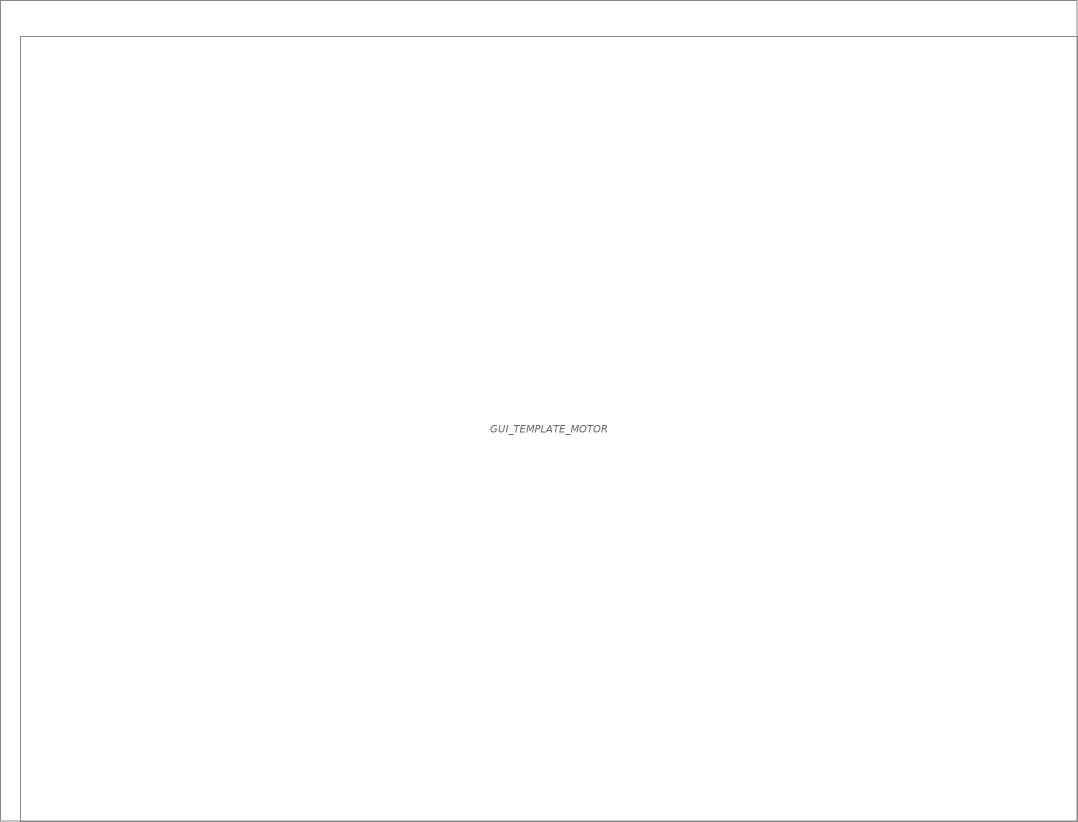
VISUALIZATION GUI_TEST_STEPPER_SHUTTER  // 1078x822
    Frame (20,36 1058x786)
        shows GUI_TEMPLATE_MOTOR(m_Instance := MAIN.nott_ics.Shutters.Test_Shutter)
END_VISUALIZATION

(* stored: Version 1.1.0.1, ProductVersion 3.1.4024.14
   Visu GUI_TEST_STEPPER_SHUTTER: Id {e1b82f2b-1971-4bac-9783-add930f3ed42} *)
